//-----------------------------------------------------------------------------------------
//
//                  				ST_HMI_Footer
//
//							Structure datas pied de page HMI 			
//-----------------------------------------------------------------------------------------
//
//Auteur: G.GOETZ
//Création: 21.01.2026
//Dernière modification : 21.01.2026 (G.GOETZ)
//       			
//-----------------------------------------------------------------------------------------
//
//     							Liste des modifications  	
//
// 21.01.2026 (G.GOETZ) -> Création		
//-----------------------------------------------------------------------------------------

TYPE ST_HMI_Footer :
STRUCT
	
	(** SETUP INT **)
		ix1 : INT ; // ?
	
	(** SETUP FLAG **)
		bx1 : BOOL ; // ?

	(** PROCESS INT **)
		iy1 : INT ; // ?
	
	(** PROCESS FLAG **)
		by1 : BOOL ; // ?
	
END_STRUCT
END_TYPE

(* stored: Version 1.1.0.1, ProductVersion 3.1.4026.17
   DUT ST_HMI_Footer: Id {c1b56779-9cea-4fe1-8728-e68fe92bdcbd} *)
